Universal Robots PolyScope program: testDoubleSensorAdaptiveGrip.urp

Program testDoubleSensorAdaptiveGrip (installation=20240827 directory=/programs createdIn=5.15.1 lastSavedIn=5.15.1 robotSerialNumber=20245500285)
Calibrated DH parameters: a=[0.000097, -0.210459, -0.026602, 0.000137, 0.000078, 0]; d=[0.162601, 254.180657, -54.076236, -199.970743, 0.099615, 0.099684]; alpha=[1.569796, -0.001455, 0.001957, 1.570525, -1.571561, 0]; deltaTheta=[0, -1.053331, 8.839472, -1.50296, 0.000002, 0]
InitVariablesNode
Robot Program (runOnlyOnce=true)
  Script: usb = rpc_factory("xmlrpc","http://192.168.1.7:9120/RPC2")
  counter := 0
  Loop Forever
    Script: usb.open()
    SuppressedNode
      Halt
    Wait Sleep waitTime=0.5
    Popup Message (haltProgram=false message=12 inputType=Text)
    MoveJ speed 60 deg/s, acceleration 80 deg/s^2 (useActiveTCP=true) feature=Base
      Waypoint 路点_1: TCP in base x=180.602 y=-555.421 z=190.206 mm, rx=-2.249 ry=-2.1664 rz=0.0591 rad; joints [95.91, -77.938, 92.238, -104.843, -92.374, 98.223] deg; TCP offset x=-0.17 y=0 z=192.95 mm, rx=0 ry=0 rz=0 rad
    Script: usb.adaptiveClose()
    var_1 := get_actual_tcp_pose()
    Script: var_1[2]=var_1[2]+0.05
    Popup Message (haltProgram=false message=12 inputType=Text)
    MoveL speed 250 mm/s, acceleration 1200 mm/s^2 (useActiveTCP=true) feature=Base
      Waypoint Variable (Variable): variable=var_1
    MoveJ speed 60 deg/s, acceleration 80 deg/s^2 (useActiveTCP=true) feature=Base
      Waypoint 路点_1: TCP in base x=180.602 y=-555.421 z=190.206 mm, rx=-2.249 ry=-2.1664 rz=0.0591 rad; joints [95.91, -77.938, 92.238, -104.843, -92.374, 98.223] deg
    Script: counter=counter+1
